            CASE ix OF
	0: getUint32 := data.ix00; (*Return index 0 for the data struct*)
	1: getUint32 := data.ix01; (*Return index 1 for the data struct*)
	2: getUint32 := data.ix02; (*Return index 2 for the data struct*)
	3: getUint32 := data.ix03; (*Return index 3 for the data struct*)
	4: getUint32 := data.ix04; (*Return index 4 for the data struct*)
	5: getUint32 := data.ix05; (*Return index 5 for the data struct*)
	6: getUint32 := data.ix06; (*Return index 6 for the data struct*)
	7: getUint32 := data.ix07; (*Return index 7 for the data struct*)
	8: getUint32 := data.ix08; (*Return index 8 for the data struct*)
	9: getUint32 := data.ix09; (*Return index 9 for the data struct*)
	10: getUint32 := data.ix10; (*Return index 10 for the data struct*)
	11: getUint32 := data.ix11; (*Return index 11 for the data struct*)
	12: getUint32 := data.ix12; (*Return index 12 for the data struct*)
	13: getUint32 := data.ix13; (*Return index 13 for the data struct*)
	14: getUint32 := data.ix14; (*Return index 14 for the data struct*)
	15: getUint32 := data.ix15; (*Return index 15 for the data struct*)
	16: getUint32 := data.ix16; (*Return index 16 for the data struct*)
	17: getUint32 := data.ix17; (*Return index 17 for the data struct*)
	18: getUint32 := data.ix18; (*Return index 18 for the data struct*)
	19: getUint32 := data.ix19; (*Return index 19 for the data struct*)
	20: getUint32 := data.ix20; (*Return index 20 for the data struct*)
	21: getUint32 := data.ix21; (*Return index 21 for the data struct*)
	22: getUint32 := data.ix22; (*Return index 22 for the data struct*)
	23: getUint32 := data.ix23; (*Return index 23 for the data struct*)
	24: getUint32 := data.ix24; (*Return index 24 for the data struct*)
	25: getUint32 := data.ix25; (*Return index 25 for the data struct*)
	26: getUint32 := data.ix26; (*Return index 26 for the data struct*)
	27: getUint32 := data.ix27; (*Return index 27 for the data struct*)
	28: getUint32 := data.ix28; (*Return index 28 for the data struct*)
	29: getUint32 := data.ix29; (*Return index 29 for the data struct*)
	30: getUint32 := data.ix30; (*Return index 30 for the data struct*)
	31: getUint32 := data.ix31; (*Return index 31 for the data struct*)
ELSE
	(*Index is invalid, return initial function value*)
	RETURN;
END_CASE
RETURN;

          
END_FUNCTION

FUNCTION getUlint32 : ULINT
  VAR_INPUT
    data : ULINT32;  (* Data to work on *)
    ix : USINT;  (* Index to retrieve *)
  END_VAR

            CASE ix OF
	0: getUlint32 := data.ix00; (*Return index 0 for the data struct*)
	1: getUlint32 := data.ix01; (*Return index 1 for the data struct*)
	2: getUlint32 := data.ix02; (*Return index 2 for the data struct*)
	3: getUlint32 := data.ix03; (*Return index 3 for the data struct*)
	4: getUlint32 := data.ix04; (*Return index 4 for the data struct*)
	5: getUlint32 := data.ix05; (*Return index 5 for the data struct*)
	6: getUlint32 := data.ix06; (*Return index 6 for the data struct*)
	7: getUlint32 := data.ix07; (*Return index 7 for the data struct*)
	8: getUlint32 := data.ix08; (*Return index 8 for the data struct*)
	9: getUlint32 := data.ix09; (*Return index 9 for the data struct*)
	10: getUlint32 := data.ix10; (*Return index 10 for the data struct*)
	11: getUlint32 := data.ix11; (*Return index 11 for the data struct*)
	12: getUlint32 := data.ix12; (*Return index 12 for the data struct*)
	13: getUlint32 := data.ix13; (*Return index 13 for the data struct*)
	14: getUlint32 := data.ix14; (*Return index 14 for the data struct*)
	15: getUlint32 := data.ix15; (*Return index 15 for the data struct*)
	16: getUlint32 := data.ix16; (*Return index 16 for the data struct*)
	17: getUlint32 := data.ix17; (*Return index 17 for the data struct*)
	18: getUlint32 := data.ix18; (*Return index 18 for the data struct*)
	19: getUlint32 := data.ix19; (*Return index 19 for the data struct*)
	20: getUlint32 := data.ix20; (*Return index 20 for the data struct*)
	21: getUlint32 := data.ix21; (*Return index 21 for the data struct*)
	22: getUlint32 := data.ix22; (*Return index 22 for the data struct*)
	23: getUlint32 := data.ix23; (*Return index 23 for the data struct*)
	24: getUlint32 := data.ix24; (*Return index 24 for the data struct*)
	25: getUlint32 := data.ix25; (*Return index 25 for the data struct*)
	26: getUlint32 := data.ix26; (*Return index 26 for the data struct*)
	27: getUlint32 := data.ix27; (*Return index 27 for the data struct*)
	28: getUlint32 := data.ix28; (*Return index 28 for the data struct*)
	29: getUlint32 := data.ix29; (*Return index 29 for the data struct*)
	30: getUlint32 := data.ix30; (*Return index 30 for the data struct*)
	31: getUlint32 := data.ix31; (*Return index 31 for the data struct*)
ELSE
	(*Index is invalid, return initial function value*)
	RETURN;
END_CASE
RETURN;

          
END_FUNCTION

FUNCTION getUsint32 : USINT
  VAR_INPUT
    data : USINT32;  (* Data to work on *)
    ix : USINT;  (* Index to retrieve *)
  END_VAR

            CASE ix OF
	0: getUsint32 := data.ix00; (*Return index 0 for the data struct*)
	1: getUsint32 := data.ix01; (*Return index 1 for the data struct*)
	2: getUsint32 := data.ix02; (*Return index 2 for the data struct*)
	3: getUsint32 := data.ix03; (*Return index 3 for the data struct*)
	4: getUsint32 := data.ix04; (*Return index 4 for the data struct*)
	5: getUsint32 := data.ix05; (*Return index 5 for the data struct*)
	6: getUsint32 := data.ix06; (*Return index 6 for the data struct*)
	7: getUsint32 := data.ix07; (*Return index 7 for the data struct*)
	8: getUsint32 := data.ix08; (*Return index 8 for the data struct*)
	9: getUsint32 := data.ix09; (*Return index 9 for the data struct*)
	10: getUsint32 := data.ix10; (*Return index 10 for the data struct*)
	11: getUsint32 := data.ix11; (*Return index 11 for the data struct*)
	12: getUsint32 := data.ix12; (*Return index 12 for the data struct*)
	13: getUsint32 := data.ix13; (*Return index 13 for the data struct*)
	14: getUsint32 := data.ix14; (*Return index 14 for the data struct*)
	15: getUsint32 := data.ix15; (*Return index 15 for the data struct*)
	16: getUsint32 := data.ix16; (*Return index 16 for the data struct*)
	17: getUsint32 := data.ix17; (*Return index 17 for the data struct*)
	18: getUsint32 := data.ix18; (*Return index 18 for the data struct*)
	19: getUsint32 := data.ix19; (*Return index 19 for the data struct*)
	20: getUsint32 := data.ix20; (*Return index 20 for the data struct*)
	21: getUsint32 := data.ix21; (*Return index 21 for the data struct*)
	22: getUsint32 := data.ix22; (*Return index 22 for the data struct*)
	23: getUsint32 := data.ix23; (*Return index 23 for the data struct*)
	24: getUsint32 := data.ix24; (*Return index 24 for the data struct*)
	25: getUsint32 := data.ix25; (*Return index 25 for the data struct*)
	26: getUsint32 := data.ix26; (*Return index 26 for the data struct*)
	27: getUsint32 := data.ix27; (*Return index 27 for the data struct*)
	28: getUsint32 := data.ix28; (*Return index 28 for the data struct*)
	29: getUsint32 := data.ix29; (*Return index 29 for the data struct*)
	30: getUsint32 := data.ix30; (*Return index 30 for the data struct*)
	31: getUsint32 := data.ix31; (*Return index 31 for the data struct*)
ELSE
	(*Index is invalid, return initial function value*)
	RETURN;
END_CASE
RETURN;

          
END_FUNCTION

FUNCTION getWord32 : WORD
  VAR_INPUT
    data : WORD32;  (* Data to work on *)
    ix : USINT;  (* Index to retrieve *)
  END_VAR

            CASE ix OF
	0: getWord32 := data.ix00; (*Return index 0 for the data struct*)
	1: getWord32 := data.ix01; (*Return index 1 for the data struct*)
	2: getWord32 := data.ix02; (*Return index 2 for the data struct*)
	3: getWord32 := data.ix03; (*Return index 3 for the data struct*)
	4: getWord32 := data.ix04; (*Return index 4 for the data struct*)
	5: getWord32 := data.ix05; (*Return index 5 for the data struct*)
	6: getWord32 := data.ix06; (*Return index 6 for the data struct*)
	7: getWord32 := data.ix07; (*Return index 7 for the data struct*)
	8: getWord32 := data.ix08; (*Return index 8 for the data struct*)
	9: getWord32 := data.ix09; (*Return index 9 for the data struct*)
	10: getWord32 := data.ix10; (*Return index 10 for the data struct*)
	11: getWord32 := data.ix11; (*Return index 11 for the data struct*)
	12: getWord32 := data.ix12; (*Return index 12 for the data struct*)
	13: getWord32 := data.ix13; (*Return index 13 for the data struct*)
	14: getWord32 := data.ix14; (*Return index 14 for the data struct*)
	15: getWord32 := data.ix15; (*Return index 15 for the data struct*)
	16: getWord32 := data.ix16; (*Return index 16 for the data struct*)
	17: getWord32 := data.ix17; (*Return index 17 for the data struct*)
	18: getWord32 := data.ix18; (*Return index 18 for the data struct*)
	19: getWord32 := data.ix19; (*Return index 19 for the data struct*)
	20: getWord32 := data.ix20; (*Return index 20 for the data struct*)
	21: getWord32 := data.ix21; (*Return index 21 for the data struct*)
	22: getWord32 := data.ix22; (*Return index 22 for the data struct*)
	23: getWord32 := data.ix23; (*Return index 23 for the data struct*)
	24: getWord32 := data.ix24; (*Return index 24 for the data struct*)
	25: getWord32 := data.ix25; (*Return index 25 for the data struct*)
	26: getWord32 := data.ix26; (*Return index 26 for the data struct*)
	27: getWord32 := data.ix27; (*Return index 27 for the data struct*)
	28: getWord32 := data.ix28; (*Return index 28 for the data struct*)
	29: getWord32 := data.ix29; (*Return index 29 for the data struct*)
	30: getWord32 := data.ix30; (*Return index 30 for the data struct*)
	31: getWord32 := data.ix31; (*Return index 31 for the data struct*)
ELSE
	(*Index is invalid, return initial function value*)
	RETURN;
END_CASE
RETURN;

          
END_FUNCTION

FUNCTION getWstring32 : WSTRING
  VAR_INPUT
    data : WSTRING32;  (* Data to work on *)
    ix : USINT;  (* Index to retrieve *)
  END_VAR

            CASE ix OF
	0: getWstring32 := data.ix00; (*Return index 0 for the data struct*)
	1: getWstring32 := data.ix01; (*Return index 1 for the data struct*)
	2: getWstring32 := data.ix02; (*Return index 2 for the data struct*)
	3: getWstring32 := data.ix03; (*Return index 3 for the data struct*)
	4: getWstring32 := data.ix04; (*Return index 4 for the data struct*)
	5: getWstring32 := data.ix05; (*Return index 5 for the data struct*)
	6: getWstring32 := data.ix06; (*Return index 6 for the data struct*)
	7: getWstring32 := data.ix07; (*Return index 7 for the data struct*)
	8: getWstring32 := data.ix08; (*Return index 8 for the data struct*)
	9: getWstring32 := data.ix09; (*Return index 9 for the data struct*)
	10: getWstring32 := data.ix10; (*Return index 10 for the data struct*)
	11: getWstring32 := data.ix11; (*Return index 11 for the data struct*)
	12: getWstring32 := data.ix12; (*Return index 12 for the data struct*)
	13: getWstring32 := data.ix13; (*Return index 13 for the data struct*)
	14: getWstring32 := data.ix14; (*Return index 14 for the data struct*)
	15: getWstring32 := data.ix15; (*Return index 15 for the data struct*)
	16: getWstring32 := data.ix16; (*Return index 16 for the data struct*)
	17: getWstring32 := data.ix17; (*Return index 17 for the data struct*)
	18: getWstring32 := data.ix18; (*Return index 18 for the data struct*)
	19: getWstring32 := data.ix19; (*Return index 19 for the data struct*)
	20: getWstring32 := data.ix20; (*Return index 20 for the data struct*)
	21: getWstring32 := data.ix21; (*Return index 21 for the data struct*)
	22: getWstring32 := data.ix22; (*Return index 22 for the data struct*)
	23: getWstring32 := data.ix23; (*Return index 23 for the data struct*)
	24: getWstring32 := data.ix24; (*Return index 24 for the data struct*)
	25: getWstring32 := data.ix25; (*Return index 25 for the data struct*)
	26: getWstring32 := data.ix26; (*Return index 26 for the data struct*)
	27: getWstring32 := data.ix27; (*Return index 27 for the data struct*)
	28: getWstring32 := data.ix28; (*Return index 28 for the data struct*)
	29: getWstring32 := data.ix29; (*Return index 29 for the data struct*)
	30: getWstring32 := data.ix30; (*Return index 30 for the data struct*)
	31: getWstring32 := data.ix31; (*Return index 31 for the data struct*)
ELSE
	(*Index is invalid, return initial function value*)
	RETURN;
END_CASE
RETURN;

          
END_FUNCTION

FUNCTION setBool32 : BOOL
  VAR_IN_OUT
    data : BOOL32;  (* Data to work on *)
  END_VAR
  VAR_INPUT
    ix : USINT;  (* Index to write *)
    value : BOOL;  (* Value to set to the index *)
  END_VAR

            CASE ix OF
	0: data.ix00 := value; (*Set index 0 of the data struct with the value*)
	1: data.ix01 := value; (*Set index 1 of the data struct with the value*)
	2: data.ix02 := value; (*Set index 2 of the data struct with the value*)
	3: data.ix03 := value; (*Set index 3 of the data struct with the value*)
	4: data.ix04 := value; (*Set index 4 of the data struct with the value*)
	5: data.ix05 := value; (*Set index 5 of the data struct with the value*)
	6: data.ix06 := value; (*Set index 6 of the data struct with the value*)
	7: data.ix07 := value; (*Set index 7 of the data struct with the value*)
	8: data.ix08 := value; (*Set index 8 of the data struct with the value*)
	9: data.ix09 := value; (*Set index 9 of the data struct with the value*)
	10: data.ix10 := value; (*Set index 10 of the data struct with the value*)
	11: data.ix11 := value; (*Set index 11 of the data struct with the value*)
	12: data.ix12 := value; (*Set index 12 of the data struct with the value*)
	13: data.ix13 := value; (*Set index 13 of the data struct with the value*)
	14: data.ix14 := value; (*Set index 14 of the data struct with the value*)
	15: data.ix15 := value; (*Set index 15 of the data struct with the value*)
	16: data.ix16 := value; (*Set index 16 of the data struct with the value*)
	17: data.ix17 := value; (*Set index 17 of the data struct with the value*)
	18: data.ix18 := value; (*Set index 18 of the data struct with the value*)
	19: data.ix19 := value; (*Set index 19 of the data struct with the value*)
	20: data.ix20 := value; (*Set index 20 of the data struct with the value*)
	21: data.ix21 := value; (*Set index 21 of the data struct with the value*)
	22: data.ix22 := value; (*Set index 22 of the data struct with the value*)
	23: data.ix23 := value; (*Set index 23 of the data struct with the value*)
	24: data.ix24 := value; (*Set index 24 of the data struct with the value*)
	25: data.ix25 := value; (*Set index 25 of the data struct with the value*)
	26: data.ix26 := value; (*Set index 26 of the data struct with the value*)
	27: data.ix27 := value; (*Set index 27 of the data struct with the value*)
	28: data.ix28 := value; (*Set index 28 of the data struct with the value*)
	29: data.ix29 := value; (*Set index 29 of the data struct with the value*)
	30: data.ix30 := value; (*Set index 30 of the data struct with the value*)
	31: data.ix31 := value; (*Set index 31 of the data struct with the value*)
ELSE
	(*Index is invalid, don't write anything, return false*)
	setBool32 := FALSE;
	RETURN;
END_CASE
setBool32 := TRUE;
RETURN;

          
END_FUNCTION

FUNCTION setByte32 : BOOL
  VAR_IN_OUT
    data : BYTE32;  (* Data to work on *)
  END_VAR
  VAR_INPUT
    ix : USINT;  (* Index to write *)
    value : BYTE;  (* Value to set to the index *)
  END_VAR

            CASE ix OF
	0: data.ix00 := value; (*Set index 0 of the data struct with the value*)
	1: data.ix01 := value; (*Set index 1 of the data struct with the value*)
	2: data.ix02 := value; (*Set index 2 of the data struct with the value*)
	3: data.ix03 := value; (*Set index 3 of the data struct with the value*)
	4: data.ix04 := value; (*Set index 4 of the data struct with the value*)
	5: data.ix05 := value; (*Set index 5 of the data struct with the value*)
	6: data.ix06 := value; (*Set index 6 of the data struct with the value*)
	7: data.ix07 := value; (*Set index 7 of the data struct with the value*)
	8: data.ix08 := value; (*Set index 8 of the data struct with the value*)
	9: data.ix09 := value; (*Set index 9 of the data struct with the value*)
	10: data.ix10 := value; (*Set index 10 of the data struct with the value*)
	11: data.ix11 := value; (*Set index 11 of the data struct with the value*)
	12: data.ix12 := value; (*Set index 12 of the data struct with the value*)
	13: data.ix13 := value; (*Set index 13 of the data struct with the value*)
	14: data.ix14 := value; (*Set index 14 of the data struct with the value*)
	15: data.ix15 := value; (*Set index 15 of the data struct with the value*)
	16: data.ix16 := value; (*Set index 16 of the data struct with the value*)
	17: data.ix17 := value; (*Set index 17 of the data struct with the value*)
	18: data.ix18 := value; (*Set index 18 of the data struct with the value*)
	19: data.ix19 := value; (*Set index 19 of the data struct with the value*)
	20: data.ix20 := value; (*Set index 20 of the data struct with the value*)
	21: data.ix21 := value; (*Set index 21 of the data struct with the value*)
	22: data.ix22 := value; (*Set index 22 of the data struct with the value*)
	23: data.ix23 := value; (*Set index 23 of the data struct with the value*)
	24: data.ix24 := value; (*Set index 24 of the data struct with the value*)
	25: data.ix25 := value; (*Set index 25 of the data struct with the value*)
	26: data.ix26 := value; (*Set index 26 of the data struct with the value*)
	27: data.ix27 := value; (*Set index 27 of the data struct with the value*)
	28: data.ix28 := value; (*Set index 28 of the data struct with the value*)
	29: data.ix29 := value; (*Set index 29 of the data struct with the value*)
	30: data.ix30 := value; (*Set index 30 of the data struct with the value*)
	31: data.ix31 := value; (*Set index 31 of the data struct with the value*)
ELSE
	(*Index is invalid, don't write anything, return false*)
	setByte32 := FALSE;
	RETURN;
END_CASE
setByte32 := TRUE;
RETURN;

          
END_FUNCTION

FUNCTION setDate_and_time32 : BOOL
  VAR_IN_OUT
    data : DATE_AND_TIME32;  (* Data to work on *)
  END_VAR
  VAR_INPUT
    ix : USINT;  (* Index to write *)
    value : DT;  (* Value to set to the index *)
  END_VAR

            CASE ix OF
	0: data.ix00 := value; (*Set index 0 of the data struct with the value*)
	1: data.ix01 := value; (*Set index 1 of the data struct with the value*)
	2: data.ix02 := value; (*Set index 2 of the data struct with the value*)
	3: data.ix03 := value; (*Set index 3 of the data struct with the value*)
	4: data.ix04 := value; (*Set index 4 of the data struct with the value*)
	5: data.ix05 := value; (*Set index 5 of the data struct with the value*)
	6: data.ix06 := value; (*Set index 6 of the data struct with the value*)
	7: data.ix07 := value; (*Set index 7 of the data struct with the value*)
	8: data.ix08 := value; (*Set index 8 of the data struct with the value*)
	9: data.ix09 := value; (*Set index 9 of the data struct with the value*)
	10: data.ix10 := value; (*Set index 10 of the data struct with the value*)
	11: data.ix11 := value; (*Set index 11 of the data struct with the value*)
	12: data.ix12 := value; (*Set index 12 of the data struct with the value*)
	13: data.ix13 := value; (*Set index 13 of the data struct with the value*)
	14: data.ix14 := value; (*Set index 14 of the data struct with the value*)
	15: data.ix15 := value; (*Set index 15 of the data struct with the value*)
	16: data.ix16 := value; (*Set index 16 of the data struct with the value*)
	17: data.ix17 := value; (*Set index 17 of the data struct with the value*)
	18: data.ix18 := value; (*Set index 18 of the data struct with the value*)
	19: data.ix19 := value; (*Set index 19 of the data struct with the value*)
	20: data.ix20 := value; (*Set index 20 of the data struct with the value*)
	21: data.ix21 := value; (*Set index 21 of the data struct with the value*)
	22: data.ix22 := value; (*Set index 22 of the data struct with the value*)
	23: data.ix23 := value; (*Set index 23 of the data struct with the value*)
	24: data.ix24 := value; (*Set index 24 of the data struct with the value*)
	25: data.ix25 := value; (*Set index 25 of the data struct with the value*)
	26: data.ix26 := value; (*Set index 26 of the data struct with the value*)
	27: data.ix27 := value; (*Set index 27 of the data struct with the value*)
	28: data.ix28 := value; (*Set index 28 of the data struct with the value*)
	29: data.ix29 := value; (*Set index 29 of the data struct with the value*)
	30: data.ix30 := value; (*Set index 30 of the data struct with the value*)
	31: data.ix31 := value; (*Set index 31 of the data struct with the value*)
ELSE
	(*Index is invalid, don't write anything, return false*)
	setDate_and_time32 := FALSE;
	RETURN;
END_CASE
setDate_and_time32 := TRUE;
RETURN;

          
END_FUNCTION

FUNCTION setDate32 : BOOL
  VAR_IN_OUT
    data : DATE32;  (* Data to work on *)
  END_VAR
  VAR_INPUT
    ix : USINT;  (* Index to write *)
    value : DATE;  (* Value to set to the index *)
  END_VAR

            CASE ix OF
	0: data.ix00 := value; (*Set index 0 of the data struct with the value*)
	1: data.ix01 := value; (*Set index 1 of the data struct with the value*)
	2: data.ix02 := value; (*Set index 2 of the data struct with the value*)
	3: data.ix03 := value; (*Set index 3 of the data struct with the value*)
	4: data.ix04 := value; (*Set index 4 of the data struct with the value*)
	5: data.ix05 := value; (*Set index 5 of the data struct with the value*)
	6: data.ix06 := value; (*Set index 6 of the data struct with the value*)
	7: data.ix07 := value; (*Set index 7 of the data struct with the value*)
	8: data.ix08 := value; (*Set index 8 of the data struct with the value*)
	9: data.ix09 := value; (*Set index 9 of the data struct with the value*)
	10: data.ix10 := value; (*Set index 10 of the data struct with the value*)
	11: data.ix11 := value; (*Set index 11 of the data struct with the value*)
	12: data.ix12 := value; (*Set index 12 of the data struct with the value*)
	13: data.ix13 := value; (*Set index 13 of the data struct with the value*)
	14: data.ix14 := value; (*Set index 14 of the data struct with the value*)
	15: data.ix15 := value; (*Set index 15 of the data struct with the value*)
	16: data.ix16 := value; (*Set index 16 of the data struct with the value*)
	17: data.ix17 := value; (*Set index 17 of the data struct with the value*)
	18: data.ix18 := value; (*Set index 18 of the data struct with the value*)
	19: data.ix19 := value; (*Set index 19 of the data struct with the value*)
	20: data.ix20 := value; (*Set index 20 of the data struct with the value*)
	21: data.ix21 := value; (*Set index 21 of the data struct with the value*)
	22: data.ix22 := value; (*Set index 22 of the data struct with the value*)
	23: data.ix23 := value; (*Set index 23 of the data struct with the value*)
	24: data.ix24 := value; (*Set index 24 of the data struct with the value*)
	25: data.ix25 := value; (*Set index 25 of the data struct with the value*)
	26: data.ix26 := value; (*Set index 26 of the data struct with the value*)
	27: data.ix27 := value; (*Set index 27 of the data struct with the value*)
	28: data.ix28 := value; (*Set index 28 of the data struct with the value*)
	29: data.ix29 := value; (*Set index 29 of the data struct with the value*)
	30: data.ix30 := value; (*Set index 30 of the data struct with the value*)
	31: data.ix31 := value; (*Set index 31 of the data struct with the value*)
ELSE
	(*Index is invalid, don't write anything, return false*)
	setDate32 := FALSE;
	RETURN;
END_CASE
setDate32 := TRUE;
RETURN;

          
END_FUNCTION

FUNCTION setDint32 : BOOL
  VAR_IN_OUT
    data : DINT32;  (* Data to work on *)
  END_VAR
  VAR_INPUT
    ix : USINT;  (* Index to write *)
    value : DINT;  (* Value to set to the index *)
  END_VAR

            CASE ix OF
	0: data.ix00 := value; (*Set index 0 of the data struct with the value*)
	1: data.ix01 := value; (*Set index 1 of the data struct with the value*)
	2: data.ix02 := value; (*Set index 2 of the data struct with the value*)
	3: data.ix03 := value; (*Set index 3 of the data struct with the value*)
	4: data.ix04 := value; (*Set index 4 of the data struct with the value*)
	5: data.ix05 := value; (*Set index 5 of the data struct with the value*)
	6: data.ix06 := value; (*Set index 6 of the data struct with the value*)
	7: data.ix07 := value; (*Set index 7 of the data struct with the value*)
	8: data.ix08 := value; (*Set index 8 of the data struct with the value*)
	9: data.ix09 := value; (*Set index 9 of the data struct with the value*)
	10: data.ix10 := value; (*Set index 10 of the data struct with the value*)
	11: data.ix11 := value; (*Set index 11 of the data struct with the value*)
	12: data.ix12 := value; (*Set index 12 of the data struct with the value*)
	13: data.ix13 := value; (*Set index 13 of the data struct with the value*)
	14: data.ix14 := value; (*Set index 14 of the data struct with the value*)
	15: data.ix15 := value; (*Set index 15 of the data struct with the value*)
	16: data.ix16 := value; (*Set index 16 of the data struct with the value*)
	17: data.ix17 := value; (*Set index 17 of the data struct with the value*)
	18: data.ix18 := value; (*Set index 18 of the data struct with the value*)
	19: data.ix19 := value; (*Set index 19 of the data struct with the value*)
	20: data.ix20 := value; (*Set index 20 of the data struct with the value*)
	21: data.ix21 := value; (*Set index 21 of the data struct with the value*)
	22: data.ix22 := value; (*Set index 22 of the data struct with the value*)
	23: data.ix23 := value; (*Set index 23 of the data struct with the value*)
	24: data.ix24 := value; (*Set index 24 of the data struct with the value*)
	25: data.ix25 := value; (*Set index 25 of the data struct with the value*)
	26: data.ix26 := value; (*Set index 26 of the data struct with the value*)
	27: data.ix27 := value; (*Set index 27 of the data struct with the value*)
	28: data.ix28 := value; (*Set index 28 of the data struct with the value*)
	29: data.ix29 := value; (*Set index 29 of the data struct with the value*)
	30: data.ix30 := value; (*Set index 30 of the data struct with the value*)
	31: data.ix31 := value; (*Set index 31 of the data struct with the value*)
ELSE
	(*Index is invalid, don't write anything, return false*)
	setDint32 := FALSE;
	RETURN;
END_CASE
setDint32 := TRUE;
RETURN;

          
END_FUNCTION

FUNCTION setDword32 : BOOL
  VAR_IN_OUT
    data : DWORD32;  (* Data to work on *)
  END_VAR
  VAR_INPUT
    ix : USINT;  (* Index to write *)
    value : DWORD;  (* Value to set to the index *)
  END_VAR

            CASE ix OF
	0: data.ix00 := value; (*Set index 0 of the data struct with the value*)
	1: data.ix01 := value; (*Set index 1 of the data struct with the value*)
	2: data.ix02 := value; (*Set index 2 of the data struct with the value*)
	3: data.ix03 := value; (*Set index 3 of the data struct with the value*)
	4: data.ix04 := value; (*Set index 4 of the data struct with the value*)
	5: data.ix05 := value; (*Set index 5 of the data struct with the value*)
	6: data.ix06 := value; (*Set index 6 of the data struct with the value*)
	7: data.ix07 := value; (*Set index 7 of the data struct with the value*)
	8: data.ix08 := value; (*Set index 8 of the data struct with the value*)
	9: data.ix09 := value; (*Set index 9 of the data struct with the value*)
	10: data.ix10 := value; (*Set index 10 of the data struct with the value*)
	11: data.ix11 := value; (*Set index 11 of the data struct with the value*)
	12: data.ix12 := value; (*Set index 12 of the data struct with the value*)
	13: data.ix13 := value; (*Set index 13 of the data struct with the value*)
	14: data.ix14 := value; (*Set index 14 of the data struct with the value*)
	15: data.ix15 := value; (*Set index 15 of the data struct with the value*)
	16: data.ix16 := value; (*Set index 16 of the data struct with the value*)
	17: data.ix17 := value; (*Set index 17 of the data struct with the value*)
	18: data.ix18 := value; (*Set index 18 of the data struct with the value*)
	19: data.ix19 := value; (*Set index 19 of the data struct with the value*)
	20: data.ix20 := value; (*Set index 20 of the data struct with the value*)
	21: data.ix21 := value; (*Set index 21 of the data struct with the value*)
	22: data.ix22 := value; (*Set index 22 of the data struct with the value*)
	23: data.ix23 := value; (*Set index 23 of the data struct with the value*)
	24: data.ix24 := value; (*Set index 24 of the data struct with the value*)
	25: data.ix25 := value; (*Set index 25 of the data struct with the value*)
	26: data.ix26 := value; (*Set index 26 of the data struct with the value*)
	27: data.ix27 := value; (*Set index 27 of the data struct with the value*)
	28: data.ix28 := value; (*Set index 28 of the data struct with the value*)
	29: data.ix29 := value; (*Set index 29 of the data struct with the value*)
	30: data.ix30 := value; (*Set index 30 of the data struct with the value*)
	31: data.ix31 := value; (*Set index 31 of the data struct with the value*)
ELSE
	(*Index is invalid, don't write anything, return false*)
	setDword32 := FALSE;
	RETURN;
END_CASE
setDword32 := TRUE;
RETURN;

          
END_FUNCTION

FUNCTION setInt32 : BOOL
  VAR_IN_OUT
    data : INT32;  (* Data to work on *)
  END_VAR
  VAR_INPUT
    ix : USINT;  (* Index to write *)
    value : INT;  (* Value to set to the index *)
  END_VAR

            CASE ix OF
	0: data.ix00 := value; (*Set index 0 of the data struct with the value*)
	1: data.ix01 := value; (*Set index 1 of the data struct with the value*)
	2: data.ix02 := value; (*Set index 2 of the data struct with the value*)
	3: data.ix03 := value; (*Set index 3 of the data struct with the value*)
	4: data.ix04 := value; (*Set index 4 of the data struct with the value*)
	5: data.ix05 := value; (*Set index 5 of the data struct with the value*)
	6: data.ix06 := value; (*Set index 6 of the data struct with the value*)
	7: data.ix07 := value; (*Set index 7 of the data struct with the value*)
	8: data.ix08 := value; (*Set index 8 of the data struct with the value*)
	9: data.ix09 := value; (*Set index 9 of the data struct with the value*)
	10: data.ix10 := value; (*Set index 10 of the data struct with the value*)
	11: data.ix11 := value; (*Set index 11 of the data struct with the value*)
	12: data.ix12 := value; (*Set index 12 of the data struct with the value*)
	13: data.ix13 := value; (*Set index 13 of the data struct with the value*)
	14: data.ix14 := value; (*Set index 14 of the data struct with the value*)
	15: data.ix15 := value; (*Set index 15 of the data struct with the value*)
	16: data.ix16 := value; (*Set index 16 of the data struct with the value*)
	17: data.ix17 := value; (*Set index 17 of the data struct with the value*)
	18: data.ix18 := value; (*Set index 18 of the data struct with the value*)
	19: data.ix19 := value; (*Set index 19 of the data struct with the value*)
	20: data.ix20 := value; (*Set index 20 of the data struct with the value*)
	21: data.ix21 := value; (*Set index 21 of the data struct with the value*)
	22: data.ix22 := value; (*Set index 22 of the data struct with the value*)
	23: data.ix23 := value; (*Set index 23 of the data struct with the value*)
	24: data.ix24 := value; (*Set index 24 of the data struct with the value*)
	25: data.ix25 := value; (*Set index 25 of the data struct with the value*)
	26: data.ix26 := value; (*Set index 26 of the data struct with the value*)
	27: data.ix27 := value; (*Set index 27 of the data struct with the value*)
	28: data.ix28 := value; (*Set index 28 of the data struct with the value*)
	29: data.ix29 := value; (*Set index 29 of the data struct with the value*)
	30: data.ix30 := value; (*Set index 30 of the data struct with the value*)
	31: data.ix31 := value; (*Set index 31 of the data struct with the value*)
ELSE
	(*Index is invalid, don't write anything, return false*)
	setInt32 := FALSE;
	RETURN;
END_CASE
setInt32 := TRUE;
RETURN;

          
END_FUNCTION

FUNCTION setLdate_and_time32 : BOOL
  VAR_IN_OUT
    data : LDATE_AND_TIME32;  (* Data to work on *)
  END_VAR
  VAR_INPUT
    ix : USINT;  (* Index to write *)
    value : LDATE_AND_TIME;  (* Value to set to the index *)
  END_VAR

            CASE ix OF
	0: data.ix00 := value; (*Set index 0 of the data struct with the value*)
	1: data.ix01 := value; (*Set index 1 of the data struct with the value*)
	2: data.ix02 := value; (*Set index 2 of the data struct with the value*)
	3: data.ix03 := value; (*Set index 3 of the data struct with the value*)
	4: data.ix04 := value; (*Set index 4 of the data struct with the value*)
	5: data.ix05 := value; (*Set index 5 of the data struct with the value*)
	6: data.ix06 := value; (*Set index 6 of the data struct with the value*)
	7: data.ix07 := value; (*Set index 7 of the data struct with the value*)
	8: data.ix08 := value; (*Set index 8 of the data struct with the value*)
	9: data.ix09 := value; (*Set index 9 of the data struct with the value*)
	10: data.ix10 := value; (*Set index 10 of the data struct with the value*)
	11: data.ix11 := value; (*Set index 11 of the data struct with the value*)
	12: data.ix12 := value; (*Set index 12 of the data struct with the value*)
	13: data.ix13 := value; (*Set index 13 of the data struct with the value*)
	14: data.ix14 := value; (*Set index 14 of the data struct with the value*)
	15: data.ix15 := value; (*Set index 15 of the data struct with the value*)
	16: data.ix16 := value; (*Set index 16 of the data struct with the value*)
	17: data.ix17 := value; (*Set index 17 of the data struct with the value*)
	18: data.ix18 := value; (*Set index 18 of the data struct with the value*)
	19: data.ix19 := value; (*Set index 19 of the data struct with the value*)
	20: data.ix20 := value; (*Set index 20 of the data struct with the value*)
	21: data.ix21 := value; (*Set index 21 of the data struct with the value*)
	22: data.ix22 := value; (*Set index 22 of the data struct with the value*)
	23: data.ix23 := value; (*Set index 23 of the data struct with the value*)
	24: data.ix24 := value; (*Set index 24 of the data struct with the value*)
	25: data.ix25 := value; (*Set index 25 of the data struct with the value*)
	26: data.ix26 := value; (*Set index 26 of the data struct with the value*)
	27: data.ix27 := value; (*Set index 27 of the data struct with the value*)
	28: data.ix28 := value; (*Set index 28 of the data struct with the value*)
	29: data.ix29 := value; (*Set index 29 of the data struct with the value*)
	30: data.ix30 := value; (*Set index 30 of the data struct with the value*)
	31: data.ix31 := value; (*Set index 31 of the data struct with the value*)
ELSE
	(*Index is invalid, don't write anything, return false*)
	setLdate_and_time32 := FALSE;
	RETURN;
END_CASE
setLdate_and_time32 := TRUE;
RETURN;

          
END_FUNCTION

FUNCTION setLdate32 : BOOL
  VAR_IN_OUT
    data : LDATE32;  (* Data to work on *)
  END_VAR
  VAR_INPUT
    ix : USINT;  (* Index to write *)
    value : LDATE;  (* Value to set to the index *)
  END_VAR

            CASE ix OF
	0: data.ix00 := value; (*Set index 0 of the data struct with the value*)
	1: data.ix01 := value; (*Set index 1 of the data struct with the value*)
	2: data.ix02 := value; (*Set index 2 of the data struct with the value*)
	3: data.ix03 := value; (*Set index 3 of the data struct with the value*)
	4: data.ix04 := value; (*Set index 4 of the data struct with the value*)
	5: data.ix05 := value; (*Set index 5 of the data struct with the value*)
	6: data.ix06 := value; (*Set index 6 of the data struct with the value*)
	7: data.ix07 := value; (*Set index 7 of the data struct with the value*)
	8: data.ix08 := value; (*Set index 8 of the data struct with the value*)
	9: data.ix09 := value; (*Set index 9 of the data struct with the value*)
	10: data.ix10 := value; (*Set index 10 of the data struct with the value*)
	11: data.ix11 := value; (*Set index 11 of the data struct with the value*)
	12: data.ix12 := value; (*Set index 12 of the data struct with the value*)
	13: data.ix13 := value; (*Set index 13 of the data struct with the value*)
	14: data.ix14 := value; (*Set index 14 of the data struct with the value*)
	15: data.ix15 := value; (*Set index 15 of the data struct with the value*)
	16: data.ix16 := value; (*Set index 16 of the data struct with the value*)
	17: data.ix17 := value; (*Set index 17 of the data struct with the value*)
	18: data.ix18 := value; (*Set index 18 of the data struct with the value*)
	19: data.ix19 := value; (*Set index 19 of the data struct with the value*)
	20: data.ix20 := value; (*Set index 20 of the data struct with the value*)
	21: data.ix21 := value; (*Set index 21 of the data struct with the value*)
	22: data.ix22 := value; (*Set index 22 of the data struct with the value*)
	23: data.ix23 := value; (*Set index 23 of the data struct with the value*)
	24: data.ix24 := value; (*Set index 24 of the data struct with the value*)
	25: data.ix25 := value; (*Set index 25 of the data struct with the value*)
	26: data.ix26 := value; (*Set index 26 of the data struct with the value*)
	27: data.ix27 := value; (*Set index 27 of the data struct with the value*)
	28: data.ix28 := value; (*Set index 28 of the data struct with the value*)
	29: data.ix29 := value; (*Set index 29 of the data struct with the value*)
	30: data.ix30 := value; (*Set index 30 of the data struct with the value*)
	31: data.ix31 := value; (*Set index 31 of the data struct with the value*)
ELSE
	(*Index is invalid, don't write anything, return false*)
	setLdate32 := FALSE;
	RETURN;
END_CASE
setLdate32 := TRUE;
RETURN;

          
END_FUNCTION

FUNCTION setLint32 : BOOL
  VAR_IN_OUT
    data : LINT32;  (* Data to work on *)
  END_VAR
  VAR_INPUT
    ix : USINT;  (* Index to write *)
    value : LINT;  (* Value to set to the index *)
  END_VAR

            CASE ix OF
	0: data.ix00 := value; (*Set index 0 of the data struct with the value*)
	1: data.ix01 := value; (*Set index 1 of the data struct with the value*)
	2: data.ix02 := value; (*Set index 2 of the data struct with the value*)
	3: data.ix03 := value; (*Set index 3 of the data struct with the value*)
	4: data.ix04 := value; (*Set index 4 of the data struct with the value*)
	5: data.ix05 := value; (*Set index 5 of the data struct with the value*)
	6: data.ix06 := value; (*Set index 6 of the data struct with the value*)
	7: data.ix07 := value; (*Set index 7 of the data struct with the value*)
	8: data.ix08 := value; (*Set index 8 of the data struct with the value*)
	9: data.ix09 := value; (*Set index 9 of the data struct with the value*)
	10: data.ix10 := value; (*Set index 10 of the data struct with the value*)
	11: data.ix11 := value; (*Set index 11 of the data struct with the value*)
	12: data.ix12 := value; (*Set index 12 of the data struct with the value*)
	13: data.ix13 := value; (*Set index 13 of the data struct with the value*)
	14: data.ix14 := value; (*Set index 14 of the data struct with the value*)
	15: data.ix15 := value; (*Set index 15 of the data struct with the value*)
	16: data.ix16 := value; (*Set index 16 of the data struct with the value*)
	17: data.ix17 := value; (*Set index 17 of the data struct with the value*)
	18: data.ix18 := value; (*Set index 18 of the data struct with the value*)
	19: data.ix19 := value; (*Set index 19 of the data struct with the value*)
	20: data.ix20 := value; (*Set index 20 of the data struct with the value*)
	21: data.ix21 := value; (*Set index 21 of the data struct with the value*)
	22: data.ix22 := value; (*Set index 22 of the data struct with the value*)
	23: data.ix23 := value; (*Set index 23 of the data struct with the value*)
	24: data.ix24 := value; (*Set index 24 of the data struct with the value*)
	25: data.ix25 := value; (*Set index 25 of the data struct with the value*)
	26: data.ix26 := value; (*Set index 26 of the data struct with the value*)
	27: data.ix27 := value; (*Set index 27 of the data struct with the value*)
	28: data.ix28 := value; (*Set index 28 of the data struct with the value*)
	29: data.ix29 := value; (*Set index 29 of the data struct with the value*)
	30: data.ix30 := value; (*Set index 30 of the data struct with the value*)
	31: data.ix31 := value; (*Set index 31 of the data struct with the value*)
ELSE
	(*Index is invalid, don't write anything, return false*)
	setLint32 := FALSE;
	RETURN;
END_CASE
setLint32 := TRUE;
RETURN;

          
END_FUNCTION

FUNCTION setLreal32 : BOOL
  VAR_IN_OUT
    data : LREAL32;  (* Data to work on *)
  END_VAR
  VAR_INPUT
    ix : USINT;  (* Index to write *)
    value : LREAL;  (* Value to set to the index *)
  END_VAR

            CASE ix OF
	0: data.ix00 := value; (*Set index 0 of the data struct with the value*)
	1: data.ix01 := value; (*Set index 1 of the data struct with the value*)
	2: data.ix02 := value; (*Set index 2 of the data struct with the value*)
	3: data.ix03 := value; (*Set index 3 of the data struct with the value*)
	4: data.ix04 := value; (*Set index 4 of the data struct with the value*)
	5: data.ix05 := value; (*Set index 5 of the data struct with the value*)
	6: data.ix06 := value; (*Set index 6 of the data struct with the value*)
	7: data.ix07 := value; (*Set index 7 of the data struct with the value*)
	8: data.ix08 := value; (*Set index 8 of the data struct with the value*)
	9: data.ix09 := value; (*Set index 9 of the data struct with the value*)
	10: data.ix10 := value; (*Set index 10 of the data struct with the value*)
	11: data.ix11 := value; (*Set index 11 of the data struct with the value*)
	12: data.ix12 := value; (*Set index 12 of the data struct with the value*)
	13: data.ix13 := value; (*Set index 13 of the data struct with the value*)
	14: data.ix14 := value; (*Set index 14 of the data struct with the value*)
	15: data.ix15 := value; (*Set index 15 of the data struct with the value*)
	16: data.ix16 := value; (*Set index 16 of the data struct with the value*)
	17: data.ix17 := value; (*Set index 17 of the data struct with the value*)
	18: data.ix18 := value; (*Set index 18 of the data struct with the value*)
	19: data.ix19 := value; (*Set index 19 of the data struct with the value*)
	20: data.ix20 := value; (*Set index 20 of the data struct with the value*)
	21: data.ix21 := value; (*Set index 21 of the data struct with the value*)
	22: data.ix22 := value; (*Set index 22 of the data struct with the value*)
	23: data.ix23 := value; (*Set index 23 of the data struct with the value*)
	24: data.ix24 := value; (*Set index 24 of the data struct with the value*)
	25: data.ix25 := value; (*Set index 25 of the data struct with the value*)
	26: data.ix26 := value; (*Set index 26 of the data struct with the value*)
	27: data.ix27 := value; (*Set index 27 of the data struct with the value*)
	28: data.ix28 := value; (*Set index 28 of the data struct with the value*)
	29: data.ix29 := value; (*Set index 29 of the data struct with the value*)
	30: data.ix30 := value; (*Set index 30 of the data struct with the value*)
	31: data.ix31 := value; (*Set index 31 of the data struct with the value*)
ELSE
	(*Index is invalid, don't write anything, return false*)
	setLreal32 := FALSE;
	RETURN;
END_CASE
setLreal32 := TRUE;
RETURN;

          
END_FUNCTION

FUNCTION setLtime_of_day32 : BOOL
  VAR_IN_OUT
    data : LTIME_OF_DAY32;  (* Data to work on *)
  END_VAR
  VAR_INPUT
    ix : USINT;  (* Index to write *)
    value : LTIME_OF_DAY;  (* Value to set to the index *)
  END_VAR

            CASE ix OF
	0: data.ix00 := value; (*Set index 0 of the data struct with the value*)
	1: data.ix01 := value; (*Set index 1 of the data struct with the value*)
	2: data.ix02 := value; (*Set index 2 of the data struct with the value*)
	3: data.ix03 := value; (*Set index 3 of the data struct with the value*)
	4: data.ix04 := value; (*Set index 4 of the data struct with the value*)
	5: data.ix05 := value; (*Set index 5 of the data struct with the value*)
	6: data.ix06 := value; (*Set index 6 of the data struct with the value*)
	7: data.ix07 := value; (*Set index 7 of the data struct with the value*)
	8: data.ix08 := value; (*Set index 8 of the data struct with the value*)
	9: data.ix09 := value; (*Set index 9 of the data struct with the value*)
	10: data.ix10 := value; (*Set index 10 of the data struct with the value*)
	11: data.ix11 := value; (*Set index 11 of the data struct with the value*)
	12: data.ix12 := value; (*Set index 12 of the data struct with the value*)
	13: data.ix13 := value; (*Set index 13 of the data struct with the value*)
	14: data.ix14 := value; (*Set index 14 of the data struct with the value*)
	15: data.ix15 := value; (*Set index 15 of the data struct with the value*)
	16: data.ix16 := value; (*Set index 16 of the data struct with the value*)
	17: data.ix17 := value; (*Set index 17 of the data struct with the value*)
	18: data.ix18 := value; (*Set index 18 of the data struct with the value*)
	19: data.ix19 := value; (*Set index 19 of the data struct with the value*)
	20: data.ix20 := value; (*Set index 20 of the data struct with the value*)
	21: data.ix21 := value; (*Set index 21 of the data struct with the value*)
	22: data.ix22 := value; (*Set index 22 of the data struct with the value*)
	23: data.ix23 := value; (*Set index 23 of the data struct with the value*)
	24: data.ix24 := value; (*Set index 24 of the data struct with the value*)
	25: data.ix25 := value; (*Set index 25 of the data struct with the value*)
	26: data.ix26 := value; (*Set index 26 of the data struct with the value*)
	27: data.ix27 := value; (*Set index 27 of the data struct with the value*)
	28: data.ix28 := value; (*Set index 28 of the data struct with the value*)
	29: data.ix29 := value; (*Set index 29 of the data struct with the value*)
	30: data.ix30 := value; (*Set index 30 of the data struct with the value*)
	31: data.ix31 := value; (*Set index 31 of the data struct with the value*)
ELSE
	(*Index is invalid, don't write anything, return false*)
	setLtime_of_day32 := FALSE;
	RETURN;
END_CASE
setLtime_of_day32 := TRUE;
RETURN;

          
END_FUNCTION

FUNCTION setLtime32 : BOOL
  VAR_IN_OUT
    data : LTIME32;  (* Data to work on *)
  END_VAR
  VAR_INPUT
    ix : USINT;  (* Index to write *)
    value : LTIME;  (* Value to set to the index *)
  END_VAR

            CASE ix OF
	0: data.ix00 := value; (*Set index 0 of the data struct with the value*)
	1: data.ix01 := value; (*Set index 1 of the data struct with the value*)
	2: data.ix02 := value; (*Set index 2 of the data struct with the value*)
	3: data.ix03 := value; (*Set index 3 of the data struct with the value*)
	4: data.ix04 := value; (*Set index 4 of the data struct with the value*)
	5: data.ix05 := value; (*Set index 5 of the data struct with the value*)
	6: data.ix06 := value; (*Set index 6 of the data struct with the value*)
	7: data.ix07 := value; (*Set index 7 of the data struct with the value*)
	8: data.ix08 := value; (*Set index 8 of the data struct with the value*)
	9: data.ix09 := value; (*Set index 9 of the data struct with the value*)
	10: data.ix10 := value; (*Set index 10 of the data struct with the value*)
	11: data.ix11 := value; (*Set index 11 of the data struct with the value*)
	12: data.ix12 := value; (*Set index 12 of the data struct with the value*)
	13: data.ix13 := value; (*Set index 13 of the data struct with the value*)
	14: data.ix14 := value; (*Set index 14 of the data struct with the value*)
	15: data.ix15 := value; (*Set index 15 of the data struct with the value*)
	16: data.ix16 := value; (*Set index 16 of the data struct with the value*)
	17: data.ix17 := value; (*Set index 17 of the data struct with the value*)
	18: data.ix18 := value; (*Set index 18 of the data struct with the value*)
	19: data.ix19 := value; (*Set index 19 of the data struct with the value*)
	20: data.ix20 := value; (*Set index 20 of the data struct with the value*)
	21: data.ix21 := value; (*Set index 21 of the data struct with the value*)
	22: data.ix22 := value; (*Set index 22 of the data struct with the value*)
	23: data.ix23 := value; (*Set index 23 of the data struct with the value*)
	24: data.ix24 := value; (*Set index 24 of the data struct with the value*)
	25: data.ix25 := value; (*Set index 25 of the data struct with the value*)
	26: data.ix26 := value; (*Set index 26 of the data struct with the value*)
	27: data.ix27 := value; (*Set index 27 of the data struct with the value*)
	28: data.ix28 := value; (*Set index 28 of the data struct with the value*)
	29: data.ix29 := value; (*Set index 29 of the data struct with the value*)
	30: data.ix30 := value; (*Set index 30 of the data struct with the value*)
	31: data.ix31 := value; (*Set index 31 of the data struct with the value*)
ELSE
	(*Index is invalid, don't write anything, return false*)
	setLtime32 := FALSE;
	RETURN;
END_CASE
setLtime32 := TRUE;
RETURN;

          
END_FUNCTION

FUNCTION setLword32 : BOOL
  VAR_IN_OUT
    data : LWORD32;  (* Data to work on *)
  END_VAR
  VAR_INPUT
    ix : USINT;  (* Index to write *)
    value : LWORD;  (* Value to set to the index *)
  END_VAR

            CASE ix OF
	0: data.ix00 := value; (*Set index 0 of the data struct with the value*)
	1: data.ix01 := value; (*Set index 1 of the data struct with the value*)
	2: data.ix02 := value; (*Set index 2 of the data struct with the value*)
	3: data.ix03 := value; (*Set index 3 of the data struct with the value*)
	4: data.ix04 := value; (*Set index 4 of the data struct with the value*)
	5: data.ix05 := value; (*Set index 5 of the data struct with the value*)
	6: data.ix06 := value; (*Set index 6 of the data struct with the value*)
	7: data.ix07 := value; (*Set index 7 of the data struct with the value*)
	8: data.ix08 := value; (*Set index 8 of the data struct with the value*)
	9: data.ix09 := value; (*Set index 9 of the data struct with the value*)
	10: data.ix10 := value; (*Set index 10 of the data struct with the value*)
	11: data.ix11 := value; (*Set index 11 of the data struct with the value*)
	12: data.ix12 := value; (*Set index 12 of the data struct with the value*)
	13: data.ix13 := value; (*Set index 13 of the data struct with the value*)
	14: data.ix14 := value; (*Set index 14 of the data struct with the value*)
	15: data.ix15 := value; (*Set index 15 of the data struct with the value*)
	16: data.ix16 := value; (*Set index 16 of the data struct with the value*)
	17: data.ix17 := value; (*Set index 17 of the data struct with the value*)
	18: data.ix18 := value; (*Set index 18 of the data struct with the value*)
	19: data.ix19 := value; (*Set index 19 of the data struct with the value*)
	20: data.ix20 := value; (*Set index 20 of the data struct with the value*)
	21: data.ix21 := value; (*Set index 21 of the data struct with the value*)
	22: data.ix22 := value; (*Set index 22 of the data struct with the value*)
	23: data.ix23 := value; (*Set index 23 of the data struct with the value*)
	24: data.ix24 := value; (*Set index 24 of the data struct with the value*)
	25: data.ix25 := value; (*Set index 25 of the data struct with the value*)
	26: data.ix26 := value; (*Set index 26 of the data struct with the value*)
	27: data.ix27 := value; (*Set index 27 of the data struct with the value*)
	28: data.ix28 := value; (*Set index 28 of the data struct with the value*)
	29: data.ix29 := value; (*Set index 29 of the data struct with the value*)
	30: data.ix30 := value; (*Set index 30 of the data struct with the value*)
	31: data.ix31 := value; (*Set index 31 of the data struct with the value*)
ELSE
	(*Index is invalid, don't write anything, return false*)
	setLword32 := FALSE;
	RETURN;
END_CASE
setLword32 := TRUE;
RETURN;

          
END_FUNCTION

FUNCTION setReal32 : BOOL
  VAR_IN_OUT
    data : REAL32;  (* Data to work on *)
  END_VAR
  VAR_INPUT
    ix : USINT;  (* Index to write *)
    value : REAL;  (* Value to set to the index *)
  END_VAR

            CASE ix OF
	0: data.ix00 := value; (*Set index 0 of the data struct with the value*)
	1: data.ix01 := value; (*Set index 1 of the data struct with the value*)
	2: data.ix02 := value; (*Set index 2 of the data struct with the value*)
	3: data.ix03 := value; (*Set index 3 of the data struct with the value*)
	4: data.ix04 := value; (*Set index 4 of the data struct with the value*)
	5: data.ix05 := value; (*Set index 5 of the data struct with the value*)
	6: data.ix06 := value; (*Set index 6 of the data struct with the value*)
	7: data.ix07 := value; (*Set index 7 of the data struct with the value*)
	8: data.ix08 := value; (*Set index 8 of the data struct with the value*)
	9: data.ix09 := value; (*Set index 9 of the data struct with the value*)
	10: data.ix10 := value; (*Set index 10 of the data struct with the value*)
	11: data.ix11 := value; (*Set index 11 of the data struct with the value*)
	12: data.ix12 := value; (*Set index 12 of the data struct with the value*)
	13: data.ix13 := value; (*Set index 13 of the data struct with the value*)
	14: data.ix14 := value; (*Set index 14 of the data struct with the value*)
	15: data.ix15 := value; (*Set index 15 of the data struct with the value*)
	16: data.ix16 := value; (*Set index 16 of the data struct with the value*)
	17: data.ix17 := value; (*Set index 17 of the data struct with the value*)
	18: data.ix18 := value; (*Set index 18 of the data struct with the value*)
	19: data.ix19 := value; (*Set index 19 of the data struct with the value*)
	20: data.ix20 := value; (*Set index 20 of the data struct with the value*)
	21: data.ix21 := value; (*Set index 21 of the data struct with the value*)
	22: data.ix22 := value; (*Set index 22 of the data struct with the value*)
	23: data.ix23 := value; (*Set index 23 of the data struct with the value*)
	24: data.ix24 := value; (*Set index 24 of the data struct with the value*)
	25: data.ix25 := value; (*Set index 25 of the data struct with the value*)
	26: data.ix26 := value; (*Set index 26 of the data struct with the value*)
	27: data.ix27 := value; (*Set index 27 of the data struct with the value*)
	28: data.ix28 := value; (*Set index 28 of the data struct with the value*)
	29: data.ix29 := value; (*Set index 29 of the data struct with the value*)
	30: data.ix30 := value; (*Set index 30 of the data struct with the value*)
	31: data.ix31 := value; (*Set index 31 of the data struct with the value*)
ELSE
	(*Index is invalid, don't write anything, return false*)
	setReal32 := FALSE;
	RETURN;
END_CASE
setReal32 := TRUE;
RETURN;

          
END_FUNCTION

FUNCTION setSint32 : BOOL
  VAR_IN_OUT
    data : SINT32;  (* Data to work on *)
  END_VAR
  VAR_INPUT
    ix : USINT;  (* Index to write *)
    value : SINT;  (* Value to set to the index *)
  END_VAR

            CASE ix OF
	0: data.ix00 := value; (*Set index 0 of the data struct with the value*)
	1: data.ix01 := value; (*Set index 1 of the data struct with the value*)
	2: data.ix02 := value; (*Set index 2 of the data struct with the value*)
	3: data.ix03 := value; (*Set index 3 of the data struct with the value*)
	4: data.ix04 := value; (*Set index 4 of the data struct with the value*)
	5: data.ix05 := value; (*Set index 5 of the data struct with the value*)
	6: data.ix06 := value; (*Set index 6 of the data struct with the value*)
	7: data.ix07 := value; (*Set index 7 of the data struct with the value*)
	8: data.ix08 := value; (*Set index 8 of the data struct with the value*)
	9: data.ix09 := value; (*Set index 9 of the data struct with the value*)
	10: data.ix10 := value; (*Set index 10 of the data struct with the value*)
	11: data.ix11 := value; (*Set index 11 of the data struct with the value*)
	12: data.ix12 := value; (*Set index 12 of the data struct with the value*)
	13: data.ix13 := value; (*Set index 13 of the data struct with the value*)
	14: data.ix14 := value; (*Set index 14 of the data struct with the value*)
	15: data.ix15 := value; (*Set index 15 of the data struct with the value*)
	16: data.ix16 := value; (*Set index 16 of the data struct with the value*)
	17: data.ix17 := value; (*Set index 17 of the data struct with the value*)
	18: data.ix18 := value; (*Set index 18 of the data struct with the value*)
	19: data.ix19 := value; (*Set index 19 of the data struct with the value*)
	20: data.ix20 := value; (*Set index 20 of the data struct with the value*)
	21: data.ix21 := value; (*Set index 21 of the data struct with the value*)
	22: data.ix22 := value; (*Set index 22 of the data struct with the value*)
	23: data.ix23 := value; (*Set index 23 of the data struct with the value*)
	24: data.ix24 := value; (*Set index 24 of the data struct with the value*)
	25: data.ix25 := value; (*Set index 25 of the data struct with the value*)
	26: data.ix26 := value; (*Set index 26 of the data struct with the value*)
	27: data.ix27 := value; (*Set index 27 of the data struct with the value*)
	28: data.ix28 := value; (*Set index 28 of the data struct with the value*)
	29: data.ix29 := value; (*Set index 29 of the data struct with the value*)
	30: data.ix30 := value; (*Set index 30 of the data struct with the value*)
	31: data.ix31 := value; (*Set index 31 of the data struct with the value*)
ELSE
	(*Index is invalid, don't write anything, return false*)
	setSint32 := FALSE;
	RETURN;
END_CASE
setSint32 := TRUE;
RETURN;

          
END_FUNCTION

FUNCTION setString32 : BOOL
  VAR_IN_OUT
    data : STRING32;  (* Data to work on *)
  END_VAR
  VAR_INPUT
    ix : USINT;  (* Index to write *)
    value : STRING;  (* Value to set to the index *)
  END_VAR

            CASE ix OF
	0: data.ix00 := value; (*Set index 0 of the data struct with the value*)
	1: data.ix01 := value; (*Set index 1 of the data struct with the value*)
	2: data.ix02 := value; (*Set index 2 of the data struct with the value*)
	3: data.ix03 := value; (*Set index 3 of the data struct with the value*)
	4: data.ix04 := value; (*Set index 4 of the data struct with the value*)
	5: data.ix05 := value; (*Set index 5 of the data struct with the value*)
	6: data.ix06 := value; (*Set index 6 of the data struct with the value*)
	7: data.ix07 := value; (*Set index 7 of the data struct with the value*)
	8: data.ix08 := value; (*Set index 8 of the data struct with the value*)
	9: data.ix09 := value; (*Set index 9 of the data struct with the value*)
	10: data.ix10 := value; (*Set index 10 of the data struct with the value*)
	11: data.ix11 := value; (*Set index 11 of the data struct with the value*)
	12: data.ix12 := value; (*Set index 12 of the data struct with the value*)
	13: data.ix13 := value; (*Set index 13 of the data struct with the value*)
	14: data.ix14 := value; (*Set index 14 of the data struct with the value*)
	15: data.ix15 := value; (*Set index 15 of the data struct with the value*)
	16: data.ix16 := value; (*Set index 16 of the data struct with the value*)
	17: data.ix17 := value; (*Set index 17 of the data struct with the value*)
	18: data.ix18 := value; (*Set index 18 of the data struct with the value*)
	19: data.ix19 := value; (*Set index 19 of the data struct with the value*)
	20: data.ix20 := value; (*Set index 20 of the data struct with the value*)
	21: data.ix21 := value; (*Set index 21 of the data struct with the value*)
	22: data.ix22 := value; (*Set index 22 of the data struct with the value*)
	23: data.ix23 := value; (*Set index 23 of the data struct with the value*)
	24: data.ix24 := value; (*Set index 24 of the data struct with the value*)
	25: data.ix25 := value; (*Set index 25 of the data struct with the value*)
	26: data.ix26 := value; (*Set index 26 of the data struct with the value*)
	27: data.ix27 := value; (*Set index 27 of the data struct with the value*)
	28: data.ix28 := value; (*Set index 28 of the data struct with the value*)
	29: data.ix29 := value; (*Set index 29 of the data struct with the value*)
	30: data.ix30 := value; (*Set index 30 of the data struct with the value*)
	31: data.ix31 := value; (*Set index 31 of the data struct with the value*)
ELSE
	(*Index is invalid, don't write anything, return false*)
	setString32 := FALSE;
	RETURN;
END_CASE
setString32 := TRUE;
RETURN;

          
END_FUNCTION

FUNCTION setTime_of_day32 : BOOL
  VAR_IN_OUT
    data : TIME_OF_DAY32;  (* Data to work on *)
  END_VAR
  VAR_INPUT
    ix : USINT;  (* Index to write *)
    value : TOD;  (* Value to set to the index *)
  END_VAR

            CASE ix OF
	0: data.ix00 := value; (*Set index 0 of the data struct with the value*)
	1: data.ix01 := value; (*Set index 1 of the data struct with the value*)
	2: data.ix02 := value; (*Set index 2 of the data struct with the value*)
	3: data.ix03 := value; (*Set index 3 of the data struct with the value*)
	4: data.ix04 := value; (*Set index 4 of the data struct with the value*)
	5: data.ix05 := value; (*Set index 5 of the data struct with the value*)
	6: data.ix06 := value; (*Set index 6 of the data struct with the value*)
	7: data.ix07 := value; (*Set index 7 of the data struct with the value*)
	8: data.ix08 := value; (*Set index 8 of the data struct with the value*)
	9: data.ix09 := value; (*Set index 9 of the data struct with the value*)
	10: data.ix10 := value; (*Set index 10 of the data struct with the value*)
	11: data.ix11 := value; (*Set index 11 of the data struct with the value*)
	12: data.ix12 := value; (*Set index 12 of the data struct with the value*)
	13: data.ix13 := value; (*Set index 13 of the data struct with the value*)
	14: data.ix14 := value; (*Set index 14 of the data struct with the value*)
	15: data.ix15 := value; (*Set index 15 of the data struct with the value*)
	16: data.ix16 := value; (*Set index 16 of the data struct with the value*)
	17: data.ix17 := value; (*Set index 17 of the data struct with the value*)
	18: data.ix18 := value; (*Set index 18 of the data struct with the value*)
	19: data.ix19 := value; (*Set index 19 of the data struct with the value*)
	20: data.ix20 := value; (*Set index 20 of the data struct with the value*)
	21: data.ix21 := value; (*Set index 21 of the data struct with the value*)
	22: data.ix22 := value; (*Set index 22 of the data struct with the value*)
	23: data.ix23 := value; (*Set index 23 of the data struct with the value*)
	24: data.ix24 := value; (*Set index 24 of the data struct with the value*)
	25: data.ix25 := value; (*Set index 25 of the data struct with the value*)
	26: data.ix26 := value; (*Set index 26 of the data struct with the value*)
	27: data.ix27 := value; (*Set index 27 of the data struct with the value*)
	28: data.ix28 := value; (*Set index 28 of the data struct with the value*)
	29: data.ix29 := value; (*Set index 29 of the data struct with the value*)
	30: data.ix30 := value; (*Set index 30 of the data struct with the value*)
	31: data.ix31 := value; (*Set index 31 of the data struct with the value*)
ELSE
	(*Index is invalid, don't write anything, return false*)
	setTime_of_day32 := FALSE;
	RETURN;
END_CASE
setTime_of_day32 := TRUE;
RETURN;

          
END_FUNCTION

FUNCTION setTime32 : BOOL
  VAR_IN_OUT
    data : TIME32;  (* Data to work on *)
  END_VAR
  VAR_INPUT
    ix : USINT;  (* Index to write *)
    value : TIME;  (* Value to set to the index *)
  END_VAR

            CASE ix OF
	0: data.ix00 := value; (*Set index 0 of the data struct with the value*)
	1: data.ix01 := value; (*Set index 1 of the data struct with the value*)
	2: data.ix02 := value; (*Set index 2 of the data struct with the value*)
	3: data.ix03 := value; (*Set index 3 of the data struct with the value*)
	4: data.ix04 := value; (*Set index 4 of the data struct with the value*)
	5: data.ix05 := value; (*Set index 5 of the data struct with the value*)
	6: data.ix06 := value; (*Set index 6 of the data struct with the value*)
	7: data.ix07 := value; (*Set index 7 of the data struct with the value*)
	8: data.ix08 := value; (*Set index 8 of the data struct with the value*)
	9: data.ix09 := value; (*Set index 9 of the data struct with the value*)
	10: data.ix10 := value; (*Set index 10 of the data struct with the value*)
	11: data.ix11 := value; (*Set index 11 of the data struct with the value*)
	12: data.ix12 := value; (*Set index 12 of the data struct with the value*)
	13: data.ix13 := value; (*Set index 13 of the data struct with the value*)
	14: data.ix14 := value; (*Set index 14 of the data struct with the value*)
	15: data.ix15 := value; (*Set index 15 of the data struct with the value*)
	16: data.ix16 := value; (*Set index 16 of the data struct with the value*)
	17: data.ix17 := value; (*Set index 17 of the data struct with the value*)
	18: data.ix18 := value; (*Set index 18 of the data struct with the value*)
	19: data.ix19 := value; (*Set index 19 of the data struct with the value*)
	20: data.ix20 := value; (*Set index 20 of the data struct with the value*)
	21: data.ix21 := value; (*Set index 21 of the data struct with the value*)
	22: data.ix22 := value; (*Set index 22 of the data struct with the value*)
	23: data.ix23 := value; (*Set index 23 of the data struct with the value*)
	24: data.ix24 := value; (*Set index 24 of the data struct with the value*)
	25: data.ix25 := value; (*Set index 25 of the data struct with the value*)
	26: data.ix26 := value; (*Set index 26 of the data struct with the value*)
	27: data.ix27 := value; (*Set index 27 of the data struct with the value*)
	28: data.ix28 := value; (*Set index 28 of the data struct with the value*)
	29: data.ix29 := value; (*Set index 29 of the data struct with the value*)
	30: data.ix30 := value; (*Set index 30 of the data struct with the value*)
	31: data.ix31 := value; (*Set index 31 of the data struct with the value*)
ELSE
	(*Index is invalid, don't write anything, return false*)
	setTime32 := FALSE;
	RETURN;
END_CASE
setTime32 := TRUE;
RETURN;

          
END_FUNCTION

FUNCTION setUdint32 : BOOL
  VAR_IN_OUT
    data : UDINT32;  (* Data to work on *)
  END_VAR
  VAR_INPUT
    ix : USINT;  (* Index to write *)
    value : UDINT;  (* Value to set to the index *)
  END_VAR

            CASE ix OF
	0: data.ix00 := value; (*Set index 0 of the data struct with the value*)
	1: data.ix01 := value; (*Set index 1 of the data struct with the value*)
	2: data.ix02 := value; (*Set index 2 of the data struct with the value*)
	3: data.ix03 := value; (*Set index 3 of the data struct with the value*)
	4: data.ix04 := value; (*Set index 4 of the data struct with the value*)
	5: data.ix05 := value; (*Set index 5 of the data struct with the value*)
	6: data.ix06 := value; (*Set index 6 of the data struct with the value*)
	7: data.ix07 := value; (*Set index 7 of the data struct with the value*)
	8: data.ix08 := value; (*Set index 8 of the data struct with the value*)
	9: data.ix09 := value; (*Set index 9 of the data struct with the value*)
	10: data.ix10 := value; (*Set index 10 of the data struct with the value*)
	11: data.ix11 := value; (*Set index 11 of the data struct with the value*)
	12: data.ix12 := value; (*Set index 12 of the data struct with the value*)
	13: data.ix13 := value; (*Set index 13 of the data struct with the value*)
	14: data.ix14 := value; (*Set index 14 of the data struct with the value*)
	15: data.ix15 := value; (*Set index 15 of the data struct with the value*)
	16: data.ix16 := value; (*Set index 16 of the data struct with the value*)
	17: data.ix17 := value; (*Set index 17 of the data struct with the value*)
	18: data.ix18 := value; (*Set index 18 of the data struct with the value*)
	19: data.ix19 := value; (*Set index 19 of the data struct with the value*)
	20: data.ix20 := value; (*Set index 20 of the data struct with the value*)
	21: data.ix21 := value; (*Set index 21 of the data struct with the value*)
	22: data.ix22 := value; (*Set index 22 of the data struct with the value*)
	23: data.ix23 := value; (*Set index 23 of the data struct with the value*)
	24: data.ix24 := value; (*Set index 24 of the data struct with the value*)
	25: data.ix25 := value; (*Set index 25 of the data struct with the value*)
	26: data.ix26 := value; (*Set index 26 of the data struct with the value*)
	27: data.ix27 := value; (*Set index 27 of the data struct with the value*)
	28: data.ix28 := value; (*Set index 28 of the data struct with the value*)
	29: data.ix29 := value; (*Set index 29 of the data struct with the value*)
	30: data.ix30 := value; (*Set index 30 of the data struct with the value*)
	31: data.ix31 := value; (*Set index 31 of the data struct with the value*)
ELSE
	(*Index is invalid, don't write anything, return false*)
	setUdint32 := FALSE;
	RETURN;
END_CASE
setUdint32 := TRUE;
RETURN;

          
END_FUNCTION

FUNCTION setUDT_Cmd32 : BOOL
  VAR_IN_OUT
    data : UDT_Cmd32;  (* Data to work on *)
  END_VAR
  VAR_INPUT
    ix : USINT;  (* Index to write *)
    value : UDT_Cmd;  (* Value to set to the index *)
  END_VAR

            CASE ix OF
	0: data.udt00 := value; (*Set index 0 of the data struct with the value*)
	1: data.udt01 := value; (*Set index 1 of the data struct with the value*)
	2: data.udt02 := value; (*Set index 2 of the data struct with the value*)
	3: data.udt03 := value; (*Set index 3 of the data struct with the value*)
	4: data.udt04 := value; (*Set index 4 of the data struct with the value*)
	5: data.udt05 := value; (*Set index 5 of the data struct with the value*)
	6: data.udt06 := value; (*Set index 6 of the data struct with the value*)
	7: data.udt07 := value; (*Set index 7 of the data struct with the value*)
	8: data.udt08 := value; (*Set index 8 of the data struct with the value*)
	9: data.udt09 := value; (*Set index 9 of the data struct with the value*)
	10: data.udt10 := value; (*Set index 10 of the data struct with the value*)
	11: data.udt11 := value; (*Set index 11 of the data struct with the value*)
	12: data.udt12 := value; (*Set index 12 of the data struct with the value*)
	13: data.udt13 := value; (*Set index 13 of the data struct with the value*)
	14: data.udt14 := value; (*Set index 14 of the data struct with the value*)
	15: data.udt15 := value; (*Set index 15 of the data struct with the value*)
	16: data.udt16 := value; (*Set index 16 of the data struct with the value*)
	17: data.udt17 := value; (*Set index 17 of the data struct with the value*)
	18: data.udt18 := value; (*Set index 18 of the data struct with the value*)
	19: data.udt19 := value; (*Set index 19 of the data struct with the value*)
	20: data.udt20 := value; (*Set index 20 of the data struct with the value*)
	21: data.udt21 := value; (*Set index 21 of the data struct with the value*)
	22: data.udt22 := value; (*Set index 22 of the data struct with the value*)
	23: data.udt23 := value; (*Set index 23 of the data struct with the value*)
	24: data.udt24 := value; (*Set index 24 of the data struct with the value*)
	25: data.udt25 := value; (*Set index 25 of the data struct with the value*)
	26: data.udt26 := value; (*Set index 26 of the data struct with the value*)
	27: data.udt27 := value; (*Set index 27 of the data struct with the value*)
	28: data.udt28 := value; (*Set index 28 of the data struct with the value*)
	29: data.udt29 := value; (*Set index 29 of the data struct with the value*)
	30: data.udt30 := value; (*Set index 30 of the data struct with the value*)
	31: data.udt31 := value; (*Set index 31 of the data struct with the value*)
ELSE
	(*Index is invalid, don't write anything, return false*)
	setUDT_Cmd32 := FALSE;
	RETURN;
END_CASE
setUDT_Cmd32 := TRUE;
RETURN;

          
END_FUNCTION

FUNCTION setUint32 : BOOL
  VAR_IN_OUT
    data : UINT32;  (* Data to work on *)
  END_VAR
  VAR_INPUT
    ix : USINT;  (* Index to write *)
    value : UINT;  (* Value to set to the index *)
  END_VAR

            CASE ix OF
	0: data.ix00 := value; (*Set index 0 of the data struct with the value*)
	1: data.ix01 := value; (*Set index 1 of the data struct with the value*)
	2: data.ix02 := value; (*Set index 2 of the data struct with the value*)
	3: data.ix03 := value; (*Set index 3 of the data struct with the value*)
	4: data.ix04 := value; (*Set index 4 of the data struct with the value*)
	5: data.ix05 := value; (*Set index 5 of the data struct with the value*)
	6: data.ix06 := value; (*Set index 6 of the data struct with the value*)
	7: data.ix07 := value; (*Set index 7 of the data struct with the value*)
	8: data.ix08 := value; (*Set index 8 of the data struct with the value*)
	9: data.ix09 := value; (*Set index 9 of the data struct with the value*)
	10: data.ix10 := value; (*Set index 10 of the data struct with the value*)
	11: data.ix11 := value; (*Set index 11 of the data struct with the value*)
	12: data.ix12 := value; (*Set index 12 of the data struct with the value*)
	13: data.ix13 := value; (*Set index 13 of the data struct with the value*)
	14: data.ix14 := value; (*Set index 14 of the data struct with the value*)
	15: data.ix15 := value; (*Set index 15 of the data struct with the value*)
	16: data.ix16 := value; (*Set index 16 of the data struct with the value*)
	17: data.ix17 := value; (*Set index 17 of the data struct with the value*)
	18: data.ix18 := value; (*Set index 18 of the data struct with the value*)
	19: data.ix19 := value; (*Set index 19 of the data struct with the value*)
	20: data.ix20 := value; (*Set index 20 of the data struct with the value*)
	21: data.ix21 := value; (*Set index 21 of the data struct with the value*)
	22: data.ix22 := value; (*Set index 22 of the data struct with the value*)
	23: data.ix23 := value; (*Set index 23 of the data struct with the value*)
	24: data.ix24 := value; (*Set index 24 of the data struct with the value*)
	25: data.ix25 := value; (*Set index 25 of the data struct with the value*)
	26: data.ix26 := value; (*Set index 26 of the data struct with the value*)
	27: data.ix27 := value; (*Set index 27 of the data struct with the value*)
	28: data.ix28 := value; (*Set index 28 of the data struct with the value*)
	29: data.ix29 := value; (*Set index 29 of the data struct with the value*)
	30: data.ix30 := value; (*Set index 30 of the data struct with the value*)
	31: data.ix31 := value; (*Set index 31 of the data struct with the value*)
ELSE
	(*Index is invalid, don't write anything, return false*)
	setUint32 := FALSE;
	RETURN;
END_CASE
setUint32 := TRUE;
RETURN;

          
END_FUNCTION

FUNCTION setUlint32 : BOOL
  VAR_IN_OUT
    data : ULINT32;  (* Data to work on *)
  END_VAR
  VAR_INPUT
    ix : USINT;  (* Index to write *)
    value : ULINT;  (* Value to set to the index *)
  END_VAR

            CASE ix OF
	0: data.ix00 := value; (*Set index 0 of the data struct with the value*)
	1: data.ix01 := value; (*Set index 1 of the data struct with the value*)
	2: data.ix02 := value; (*Set index 2 of the data struct with the value*)
	3: data.ix03 := value; (*Set index 3 of the data struct with the value*)
	4: data.ix04 := value; (*Set index 4 of the data struct with the value*)
	5: data.ix05 := value; (*Set index 5 of the data struct with the value*)
	6: data.ix06 := value; (*Set index 6 of the data struct with the value*)
	7: data.ix07 := value; (*Set index 7 of the data struct with the value*)
	8: data.ix08 := value; (*Set index 8 of the data struct with the value*)
	9: data.ix09 := value; (*Set index 9 of the data struct with the value*)
	10: data.ix10 := value; (*Set index 10 of the data struct with the value*)
	11: data.ix11 := value; (*Set index 11 of the data struct with the value*)
	12: data.ix12 := value; (*Set index 12 of the data struct with the value*)
	13: data.ix13 := value; (*Set index 13 of the data struct with the value*)
	14: data.ix14 := value; (*Set index 14 of the data struct with the value*)
	15: data.ix15 := value; (*Set index 15 of the data struct with the value*)
	16: data.ix16 := value; (*Set index 16 of the data struct with the value*)
	17: data.ix17 := value; (*Set index 17 of the data struct with the value*)
	18: data.ix18 := value; (*Set index 18 of the data struct with the value*)
	19: data.ix19 := value; (*Set index 19 of the data struct with the value*)
	20: data.ix20 := value; (*Set index 20 of the data struct with the value*)
	21: data.ix21 := value; (*Set index 21 of the data struct with the value*)
	22: data.ix22 := value; (*Set index 22 of the data struct with the value*)
	23: data.ix23 := value; (*Set index 23 of the data struct with the value*)
	24: data.ix24 := value; (*Set index 24 of the data struct with the value*)
	25: data.ix25 := value; (*Set index 25 of the data struct with the value*)
	26: data.ix26 := value; (*Set index 26 of the data struct with the value*)
	27: data.ix27 := value; (*Set index 27 of the data struct with the value*)
	28: data.ix28 := value; (*Set index 28 of the data struct with the value*)
	29: data.ix29 := value; (*Set index 29 of the data struct with the value*)
	30: data.ix30 := value; (*Set index 30 of the data struct with the value*)
	31: data.ix31 := value; (*Set index 31 of the data struct with the value*)
ELSE
	(*Index is invalid, don't write anything, return false*)
	setUlint32 := FALSE;
	RETURN;
END_CASE
setUlint32 := TRUE;
RETURN;

          
END_FUNCTION

FUNCTION setUsint32 : BOOL
  VAR_IN_OUT
    data : USINT32;  (* Data to work on *)
  END_VAR
  VAR_INPUT
    ix : USINT;  (* Index to write *)
    value : USINT;  (* Value to set to the index *)
  END_VAR

            CASE ix OF
	0: data.ix00 := value; (*Set index 0 of the data struct with the value*)
	1: data.ix01 := value; (*Set index 1 of the data struct with the value*)
	2: data.ix02 := value; (*Set index 2 of the data struct with the value*)
	3: data.ix03 := value; (*Set index 3 of the data struct with the value*)
	4: data.ix04 := value; (*Set index 4 of the data struct with the value*)
	5: data.ix05 := value; (*Set index 5 of the data struct with the value*)
	6: data.ix06 := value; (*Set index 6 of the data struct with the value*)
	7: data.ix07 := value; (*Set index 7 of the data struct with the value*)
	8: data.ix08 := value; (*Set index 8 of the data struct with the value*)
	9: data.ix09 := value; (*Set index 9 of the data struct with the value*)
	10: data.ix10 := value; (*Set index 10 of the data struct with the value*)
	11: data.ix11 := value; (*Set index 11 of the data struct with the value*)
	12: data.ix12 := value; (*Set index 12 of the data struct with the value*)
	13: data.ix13 := value; (*Set index 13 of the data struct with the value*)
	14: data.ix14 := value; (*Set index 14 of the data struct with the value*)
	15: data.ix15 := value; (*Set index 15 of the data struct with the value*)
	16: data.ix16 := value; (*Set index 16 of the data struct with the value*)
	17: data.ix17 := value; (*Set index 17 of the data struct with the value*)
	18: data.ix18 := value; (*Set index 18 of the data struct with the value*)
	19: data.ix19 := value; (*Set index 19 of the data struct with the value*)
	20: data.ix20 := value; (*Set index 20 of the data struct with the value*)
	21: data.ix21 := value; (*Set index 21 of the data struct with the value*)
	22: data.ix22 := value; (*Set index 22 of the data struct with the value*)
	23: data.ix23 := value; (*Set index 23 of the data struct with the value*)
	24: data.ix24 := value; (*Set index 24 of the data struct with the value*)
	25: data.ix25 := value; (*Set index 25 of the data struct with the value*)
	26: data.ix26 := value; (*Set index 26 of the data struct with the value*)
	27: data.ix27 := value; (*Set index 27 of the data struct with the value*)
	28: data.ix28 := value; (*Set index 28 of the data struct with the value*)
	29: data.ix29 := value; (*Set index 29 of the data struct with the value*)
	30: data.ix30 := value; (*Set index 30 of the data struct with the value*)
	31: data.ix31 := value; (*Set index 31 of the data struct with the value*)
ELSE
	(*Index is invalid, don't write anything, return false*)
	setUsint32 := FALSE;
	RETURN;
END_CASE
setUsint32 := TRUE;
RETURN;

          
END_FUNCTION

FUNCTION setWord32 : BOOL
  VAR_IN_OUT
    data : WORD32;  (* Data to work on *)
  END_VAR
  VAR_INPUT
    ix : USINT;  (* Index to write *)
    value : WORD;  (* Value to set to the index *)
  END_VAR

            CASE ix OF
	0: data.ix00 := value; (*Set index 0 of the data struct with the value*)
	1: data.ix01 := value; (*Set index 1 of the data struct with the value*)
	2: data.ix02 := value; (*Set index 2 of the data struct with the value*)
	3: data.ix03 := value; (*Set index 3 of the data struct with the value*)
	4: data.ix04 := value; (*Set index 4 of the data struct with the value*)
	5: data.ix05 := value; (*Set index 5 of the data struct with the value*)
	6: data.ix06 := value; (*Set index 6 of the data struct with the value*)
	7: data.ix07 := value; (*Set index 7 of the data struct with the value*)
	8: data.ix08 := value; (*Set index 8 of the data struct with the value*)
	9: data.ix09 := value; (*Set index 9 of the data struct with the value*)
	10: data.ix10 := value; (*Set index 10 of the data struct with the value*)
	11: data.ix11 := value; (*Set index 11 of the data struct with the value*)
	12: data.ix12 := value; (*Set index 12 of the data struct with the value*)
	13: data.ix13 := value; (*Set index 13 of the data struct with the value*)
	14: data.ix14 := value; (*Set index 14 of the data struct with the value*)
	15: data.ix15 := value; (*Set index 15 of the data struct with the value*)
	16: data.ix16 := value; (*Set index 16 of the data struct with the value*)
	17: data.ix17 := value; (*Set index 17 of the data struct with the value*)
	18: data.ix18 := value; (*Set index 18 of the data struct with the value*)
	19: data.ix19 := value; (*Set index 19 of the data struct with the value*)
	20: data.ix20 := value; (*Set index 20 of the data struct with the value*)
	21: data.ix21 := value; (*Set index 21 of the data struct with the value*)
	22: data.ix22 := value; (*Set index 22 of the data struct with the value*)
	23: data.ix23 := value; (*Set index 23 of the data struct with the value*)
	24: data.ix24 := value; (*Set index 24 of the data struct with the value*)
	25: data.ix25 := value; (*Set index 25 of the data struct with the value*)
	26: data.ix26 := value; (*Set index 26 of the data struct with the value*)
	27: data.ix27 := value; (*Set index 27 of the data struct with the value*)
	28: data.ix28 := value; (*Set index 28 of the data struct with the value*)
	29: data.ix29 := value; (*Set index 29 of the data struct with the value*)
	30: data.ix30 := value; (*Set index 30 of the data struct with the value*)
	31: data.ix31 := value; (*Set index 31 of the data struct with the value*)
ELSE
	(*Index is invalid, don't write anything, return false*)
	setWord32 := FALSE;
	RETURN;
END_CASE
setWord32 := TRUE;
RETURN;

          
END_FUNCTION

FUNCTION setWstring32 : BOOL
  VAR_IN_OUT
    data : WSTRING32;  (* Data to work on *)
  END_VAR
  VAR_INPUT
    ix : USINT;  (* Index to write *)
    value : WSTRING;  (* Value to set to the index *)
  END_VAR

            CASE ix OF
	0: data.ix00 := value; (*Set index 0 of the data struct with the value*)
	1: data.ix01 := value; (*Set index 1 of the data struct with the value*)
	2: data.ix02 := value; (*Set index 2 of the data struct with the value*)
	3: data.ix03 := value; (*Set index 3 of the data struct with the value*)
	4: data.ix04 := value; (*Set index 4 of the data struct with the value*)
	5: data.ix05 := value; (*Set index 5 of the data struct with the value*)
	6: data.ix06 := value; (*Set index 6 of the data struct with the value*)
	7: data.ix07 := value; (*Set index 7 of the data struct with the value*)
	8: data.ix08 := value; (*Set index 8 of the data struct with the value*)
	9: data.ix09 := value; (*Set index 9 of the data struct with the value*)
	10: data.ix10 := value; (*Set index 10 of the data struct with the value*)
	11: data.ix11 := value; (*Set index 11 of the data struct with the value*)
	12: data.ix12 := value; (*Set index 12 of the data struct with the value*)
	13: data.ix13 := value; (*Set index 13 of the data struct with the value*)
	14: data.ix14 := value; (*Set index 14 of the data struct with the value*)
	15: data.ix15 := value; (*Set index 15 of the data struct with the value*)
	16: data.ix16 := value; (*Set index 16 of the data struct with the value*)
	17: data.ix17 := value; (*Set index 17 of the data struct with the value*)
	18: data.ix18 := value; (*Set index 18 of the data struct with the value*)
	19: data.ix19 := value; (*Set index 19 of the data struct with the value*)
	20: data.ix20 := value; (*Set index 20 of the data struct with the value*)
	21: data.ix21 := value; (*Set index 21 of the data struct with the value*)
	22: data.ix22 := value; (*Set index 22 of the data struct with the value*)
	23: data.ix23 := value; (*Set index 23 of the data struct with the value*)
	24: data.ix24 := value; (*Set index 24 of the data struct with the value*)
	25: data.ix25 := value; (*Set index 25 of the data struct with the value*)
	26: data.ix26 := value; (*Set index 26 of the data struct with the value*)
	27: data.ix27 := value; (*Set index 27 of the data struct with the value*)
	28: data.ix28 := value; (*Set index 28 of the data struct with the value*)
	29: data.ix29 := value; (*Set index 29 of the data struct with the value*)
	30: data.ix30 := value; (*Set index 30 of the data struct with the value*)
	31: data.ix31 := value; (*Set index 31 of the data struct with the value*)
ELSE
	(*Index is invalid, don't write anything, return false*)
	setWstring32 := FALSE;
	RETURN;
END_CASE
setWstring32 := TRUE;
RETURN;

          
END_FUNCTION

PROGRAM working_with_bool_struct_arrays
  VAR
    bools : BOOL32 := (ix00 := FALSE, ix01 := TRUE, ix02 := FALSE, ix03 := TRUE);  (* Boolean 32 array initialized with some values *)
    resultBool : BOOL;  (* Corresponds to index 1 of bools struct array *)
    currentBool : BOOL;  (* Used to store current iterated data *)
    movedBools : BOOL32;  (* bools struct array copied to this struct array *)
    invertedBools : BOOL32;  (* bools struct array copied and inverted to this struct array *)
    initBools : BOOL32;  (* Boolean struct array initialized with TRUE values *)
    i : USINT;  (* Iterator *)
  END_VAR

                    // WORKING WITH BOOLEAN STRUCT ARRAYS

//This returns index 1 of the struct
resultBool := getBool32(bools, 1);

//This will copy over the struct array to another array
//movedBools := bools;
// OR
FOR i:=0 TO 31 DO
	setBool32(movedBools, i, getBool32(bools, i));
END_FOR

//This will initialize/reset/fill the struct array with some values
FOR i:=0 TO 31 DO
	setBool32(initBools, i, TRUE);
END_FOR

//This will copy over the struct array to another array and do some extra logic
FOR i:=0 TO 31 DO
	currentBool := getBool32(bools, i);
	setBool32(invertedBools, i, NOT currentBool);
END_FOR



                  
END_PROGRAM

PROGRAM working_with_number_struct_arrays
  VAR
    nums : INT32 := (ix00 := -1, ix01 := 0, ix02 := 95, ix03 := 37);  (* INTEGER 32 array initialized with some values *)
    resultNum : INT;  (* Corresponds to index 1 of nums struct array *)
    currentNum : INT;  (* Used to store current iterated data *)
    movedNums : INT32;  (* nums struct array copied to this struct array *)
    incrementingNums : INT32;  (* Integer struct array that is incrementing every cycle by 1 *)
    initNums : INT32;  (* Integer struct array initialized with values from 0 - 31 *)
    i : USINT;  (* Iterator *)
  END_VAR

                    // WORKING WITH NUMBER STRUCT ARRAYS

//This returns index 1 of the struct
resultNum := getInt32(nums, 1);

//This will copy over the struct array to another array
//movedNums := nums;
// OR
FOR i:=0 TO 31 DO
	setInt32(movedNums, i, getInt32(nums, i));
END_FOR

//This will initialize/reset/fill the struct array with some values
FOR i:=0 TO 31 DO
	setInt32(initNums, i, i);
END_FOR

//This will increment every index by one each cycle
FOR i:=0 TO 31 DO
	currentNum := getInt32(incrementingNums, i);
	setInt32(incrementingNums, i, currentNum + 1);
END_FOR



                  
END_PROGRAM

PROGRAM working_with_user_datatype_struct_arrays
  VAR
    deviceCmds : UDT_Cmd32;  (* Structure array that holds all devices commands *)
    deviceStatuses : UDT_Status32;  (* Structure array that holds all devices statuses *)
    deviceCmd : UDT_Cmd;  (* Structure that holds commands only of the device currently iterated *)
    deviceStatus : UDT_Status;  (* Structure that holds status only of the device currently iterated *)
    i : USINT;  (* Iterator *)
    getCmd : getUDT_Cmd32;  (* Function block that retrieves a structure from UDT_Cmd32 struct array *)
    getStatus : getUDT_Status32;  (* Function block that retrieves a structure from UDT_Status32 struct array *)
  END_VAR

                    // WORKING WITH USER DATA TYPE STRUCT ARRAYS

FOR i:=0 TO 31 DO
	//For easier data manipulation, extract current devices commands and status
	//Now the getters must be function blocks as we cannot return as structure in iec
	getCmd(data:=deviceCmds, ix:=i);
	getStatus(data:=deviceStatuses, ix:=i);
	deviceCmd := getCmd.Out;
	deviceStatus := getStatus.Out;
	
	//If device is running, set the reference to 200
	IF deviceStatus.Running THEN
		deviceCmd.Ref := 200;
	ELSE
		deviceCmd.Ref := 0;
	END_IF
	
	//Reset device only if it has stopped
	deviceCmd.ResetCmd := deviceStatus.ResetRequired AND NOT deviceStatus.Running;
	
	//Start/Stop the device by writing to deviceCmds.udt_cmdXX from the init window*)
	deviceCmd.StartCmd := (deviceCmd.StartCmd OR deviceStatus.Running) AND NOT (deviceStatus.ResetRequired OR deviceCmd.StopCmd);
	
	//Finally write the new command data to the array
	//As we always return TRUE or FALSE we can keep this as a function
	setUDT_Cmd32(deviceCmds, i, deviceCmd);
	
END_FOR
// Manipulate the deviceStatuses from the init window
                  
END_PROGRAM

CONFIGURATION CODESYS_Control_RTE_V3_x64
  RESOURCE Application ON PLC
    TASK Task(INTERVAL := T#20ms, PRIORITY := 1);
    PROGRAM working_with_bool_struct_arrays WITH Task : working_with_bool_struct_arrays;
    PROGRAM working_with_number_struct_arrays WITH Task : working_with_number_struct_arrays;
    PROGRAM working_with_user_datatype_struct_arrays WITH Task : working_with_user_datatype_struct_arrays;
  END_RESOURCE
END_CONFIGURATION
